// TIA Portal V19 export
TYPE "Motor2Sts"
// stored: Access Published
   STRUCT
      AlarmPresence : Bool;
      RunBkwPermitted : Bool;
      RunFwdPermitted : Bool;
      Running : Bool;
   END_STRUCT;
END_TYPE
